// TwinCAT 3 PLC project PLC2
// ProgramVersion: 3.1.4026.22
// libraries:
//   Tc2_EtherCAT, * (Beckhoff Automation GmbH)
//   Tc2_Standard, * (Beckhoff Automation GmbH)
//   Tc2_System, * (Beckhoff Automation GmbH)
// project tree:
//   / PlcTask.TcTTO
//   POUs/ F_ConsumeTime.TcPOU, MAIN.TcPOU
// (motion and I/O tree: see PLC project plc1)
// real-time tasks:
//   TASK PlcTask: cycle T#10ms, priority 1, ADS port 350

CONFIGURATION PLC2
    RESOURCE PLC ON TwinCAT3
        TASK PlcTask(INTERVAL := T#10ms, PRIORITY := 1);
        PROGRAM MAIN WITH PlcTask : MAIN;
    END_RESOURCE
END_CONFIGURATION

// ---- POUs/MAIN.TcPOU
PROGRAM MAIN
VAR
END_VAR

F_ConsumeTime(75);

END_PROGRAM

// ---- POUs/F_ConsumeTime.TcPOU
FUNCTION F_ConsumeTime
VAR_INPUT
	Us		:UDINT;
END_VAR
VAR
		tCurr, tEnd : T_DCTIME64;
END_VAR

tCurr := F_GetActualDcTime64();
tEnd  := tCurr + (Us * EC_DCTIME_TICKSPERMSEC64 / 1000);
WHILE (tCurr < tEnd) DO
	tCurr := F_GetActualDcTime64();
END_WHILE

END_FUNCTION
